(* IEC 61131-3 sources: RAG_PLC/data/result/test/047, 2 files *)

(* ---- wrapped.st ---- *)
(* =========================================================
   Generated by PLC-Eval Benchmark Wrapper
   ========================================================= *)

FUNCTION_BLOCK LLM_Wrapper_FB
VAR_INPUT
	D0 : BOOL;
	D1 : BOOL;
	D2 : BOOL;
	D3 : BOOL;
	L : BOOL;
	RST : BOOL;
END_VAR

VAR_OUTPUT
	Q0 : BOOL;
	Q1 : BOOL;
	Q2 : BOOL;
	Q3 : BOOL;
END_VAR

(*@KEY@: WORKSHEET
NAME: LTCH_4
IEC_LANGUAGE: ST
*)
(* 只要 L 为 true，锁存器是透明的，D 的变化会被传递到 Q *)
(* 当然，前提是没有异步复位 *)
IF rst THEN (* 如果是异步复位，则 Q = 0 *)
	Q0 := FALSE;
	Q1 := FALSE;
	Q2 := FALSE;
	Q3 := FALSE;
ELSIF L THEN (* 锁存器是透明的 *)
	Q0 := D0;
	Q1 := D1;
	Q2 := D2;
	Q3 := D3;
END_IF;
END_FUNCTION_BLOCK

PROGRAM Auto_Proxy_Prg
  VAR
    instance : LLM_Wrapper_FB;
  END_VAR

  instance();
END_PROGRAM

CONFIGURATION Config0
  RESOURCE Res0 ON PLC
    TASK TaskMain(INTERVAL := T#20ms, PRIORITY := 0);
    PROGRAM Inst0 WITH TaskMain : Auto_Proxy_Prg;
  END_RESOURCE
END_CONFIGURATION

(* ---- raw_code.st ---- *)
VAR_INPUT
	D0 : BOOL;
	D1 : BOOL;
	D2 : BOOL;
	D3 : BOOL;
	L : BOOL;
	RST : BOOL;
END_VAR

VAR_OUTPUT
	Q0 : BOOL;
	Q1 : BOOL;
	Q2 : BOOL;
	Q3 : BOOL;
END_VAR

(*@KEY@: WORKSHEET
NAME: LTCH_4
IEC_LANGUAGE: ST
*)
(* 只要 L 为 true，锁存器是透明的，D 的变化会被传递到 Q *)
(* 当然，前提是没有异步复位 *)
IF rst THEN (* 如果是异步复位，则 Q = 0 *)
	Q0 := FALSE;
	Q1 := FALSE;
	Q2 := FALSE;
	Q3 := FALSE;
ELSIF L THEN (* 锁存器是透明的 *)
	Q0 := D0;
	Q1 := D1;
	Q2 := D2;
	Q3 := D3;
END_IF;
